// TIA Portal V18 export
// export: Created 2026-01-09T11:32:04.0126984Z, ExportSetting WithDefaults, DisplayName Totally Integrated Automation Portal, DisplayVersion V18 Update 5, DisplayName TIA Portal Openness, DisplayVersion V18 Update 5, DisplayName TIA Portal Teamcenter Gateway, DisplayVersion V18, DisplayName TIA Portal Version Control Interface, DisplayVersion V18, DisplayName SINAMICS Startdrive Advanced, DisplayVersion V18 SP2 Update 1, DisplayName SINAMICS Startdrive G110M, G120, G120C, G120D, G120P, G115D, DisplayVersion V18 SP2 Update 1, DisplayName SINAMICS Startdrive G130, G150, S120, S150, SINAMICS MV, S210, G220, S200, DisplayVersion V18 SP2 Update 1, DisplayName STEP 7 Professional, DisplayVersion V18 Update 5, DisplayName STEP 7 Safety, DisplayVersion V18, DisplayName WinCC Professional, DisplayVersion V18 Update 5
TagTable "ST_Mode"
  ST_AutoMode : Bool  (%DB[ST_SysDBNum].DBX100.0, CPU S71500-2PN_TP700, 1 s)
  ST_ManualMode : Bool  (%DB[ST_SysDBNum].DBX150.0, CPU S71500-2PN_TP700, 1 s)
  ST_StatusModeSV : Int  (%DB[ST_SysDBNum].DBW12, CPU S71500-2PN_TP700, 1 s)
  ST_StatusModePV : Int  (%DB[ST_SysDBNum].DBW14, CPU S71500-2PN_TP700, 1 s)
  Station_Sys_Cmd_ClearFlags : Bool  (PLC tag Station_Sys.Cmd.ClearFlags, %DB1060.DBX51.0, CPU S71500-2PN_TP700, 1 s)
